(* IEC 61131-3 sources: plcc/tests/fixtures/codegen, 11 files *)

(* ---- function_blocks.st ---- *)
FUNCTION_BLOCK Counter
VAR_INPUT reset : BOOL; END_VAR
VAR_OUTPUT count : INT; END_VAR
VAR cnt : INT := 0; END_VAR
    IF reset THEN cnt := 0; ELSE cnt := cnt + 1; END_IF;
    count := cnt;
END_FUNCTION_BLOCK

FUNCTION_BLOCK Doubler
VAR_INPUT val : INT; END_VAR
VAR_OUTPUT result : INT; END_VAR
    result := val + val;
END_FUNCTION_BLOCK

PROGRAM FBTest
VAR
    c1 : Counter;
    c2 : Counter;
    d : Doubler;
    sum : INT;
    doubled : INT;
END_VAR
    c1(reset := FALSE);
    c2(reset := FALSE);
    d(val := c1.count);
    sum := c1.count + c2.count;
    doubled := d.result;
END_PROGRAM

(* ---- oop.st ---- *)
FUNCTION_BLOCK Accumulator
VAR
    total : INT := 0;
END_VAR
    METHOD Add
    VAR_INPUT val : INT; END_VAR
        total := total + val;
    END_METHOD
    METHOD GetTotal : INT
        GetTotal := total;
    END_METHOD
    METHOD Reset
        total := 0;
    END_METHOD
END_FUNCTION_BLOCK

PROGRAM OOPTest
VAR
    acc : Accumulator;
    result : INT;
END_VAR
    acc.Add(val := 10);
    acc.Add(val := 20);
    acc.Add(val := 30);
    result := acc.GetTotal();
END_PROGRAM

(* ---- arithmetic.st ---- *)
PROGRAM ArithTest
VAR
    a : INT := 0;
    b : INT := 0;
    c : INT := 0;
    d : INT := 0;
    e : INT := 0;
END_VAR
    a := 10 + 5;
    b := 10 - 3;
    c := 4 * 7;
    d := 20 / 4;
    e := 17 MOD 5;
END_PROGRAM

(* ---- arrays_structs.st ---- *)
PROGRAM ArrayTest
VAR
    arr : ARRAY[0..9] OF INT;
    i : INT;
    sum : INT := 0;
    max_val : INT := 0;
END_VAR
    (* Fill array *)
    FOR i := 0 TO 9 DO
        arr[i] := (i + 1) * 10;
    END_FOR;

    (* Sum and find max *)
    sum := 0;
    max_val := arr[0];
    FOR i := 0 TO 9 DO
        sum := sum + arr[i];
        IF arr[i] > max_val THEN max_val := arr[i]; END_IF;
    END_FOR;
END_PROGRAM

(* ---- control_flow.st ---- *)
PROGRAM ControlFlow
VAR
    state : INT := 0;
    output : INT := 0;
    i : INT;
    sum : INT := 0;
END_VAR
    IF state = 0 THEN
        output := 1;
    ELSIF state = 1 THEN
        output := 2;
    ELSE
        output := 3;
    END_IF;

    sum := 0;
    FOR i := 1 TO 10 DO
        sum := sum + i;
    END_FOR;

    WHILE sum > 50 DO
        sum := sum - 10;
    END_WHILE;

    CASE state OF
        0: output := 100;
        1: output := 200;
    ELSE
        output := 0;
    END_CASE;
END_PROGRAM

(* ---- function_calls.st ---- *)
FUNCTION AddTwo : INT
VAR_INPUT
    a : INT;
    b : INT;
END_VAR
    AddTwo := a + b;
END_FUNCTION

FUNCTION Square : INT
VAR_INPUT
    x : INT;
END_VAR
    Square := x * x;
END_FUNCTION

PROGRAM CallTest
VAR
    result1 : INT;
    result2 : INT;
END_VAR
    result1 := AddTwo(3, 4);
    result2 := Square(5);
END_PROGRAM

(* ---- globals.st ---- *)
VAR_GLOBAL
    g_counter : INT;
    g_flag : BOOL;
END_VAR

PROGRAM GlobalTest
VAR
    local_copy : INT;
END_VAR
    g_counter := g_counter + 1;
    local_copy := g_counter;
END_PROGRAM

(* ---- real_fpu.st ---- *)
(* REAL arithmetic for the FPU check (crates/plcc-cli/tests/fpu.rs) and the
   Opta hardware check: results land in %M, so `img` shows them.
   %MW10 = REAL_TO_INT(((1.5 + 2.25) * (1.5 * 2.25) + 0.5) * 100) = 1316,
   %MW11 = REAL_TO_INT(SQRT(2.0) * 1000) = 1414. *)
FUNCTION Scale : REAL
VAR_INPUT
    raw : REAL;
    gain : REAL;
    offset : REAL;
END_VAR
    Scale := raw * gain + offset;
END_FUNCTION

PROGRAM Main
VAR
    a AT %MD0 : REAL := 1.5;
    b AT %MD1 : REAL := 2.25;
    sum AT %MD2 : REAL;
    prod AT %MD3 : REAL;
    q AT %MD4 : REAL;
    r AT %MW10 : INT;
    s AT %MW11 : INT;
END_VAR
    sum := a + b;
    prod := a * b;
    q := Scale(raw := sum, gain := prod, offset := 0.5);
    r := REAL_TO_INT(q * 100.0);
    s := REAL_TO_INT(SQRT(2.0) * 1000.0);
END_PROGRAM

(* ---- stdlib_conversions.st ---- *)
PROGRAM ConversionTest
VAR
    i : INT := 42;
    r : REAL;
    d : DINT;
    b : INT;
END_VAR
    r := INT_TO_REAL(i);
    d := INT_TO_DINT(i);
    b := BOOL_TO_INT(TRUE);
END_PROGRAM

(* ---- stdlib_math.st ---- *)
PROGRAM StdlibMathTest
VAR
    sq : REAL;
    ab : REAL;
    sn : REAL;
    cs : REAL;
    ex : REAL;
    lg : REAL;
    fl : REAL;
    cl : REAL;
    mn : REAL;
    mx : REAL;
    lm : REAL;
END_VAR
    sq := SQRT(25.0);
    ab := ABS(-42.0);
    sn := SIN(0.0);
    cs := COS(0.0);
    ex := EXP(0.0);
    lg := LN(1.0);
    fl := FLOOR(3.7);
    cl := CEIL(3.2);
    mn := MIN(5.0, 3.0);
    mx := MAX(5.0, 3.0);
    lm := LIMIT(0.0, -5.0, 100.0);
END_PROGRAM

(* ---- stdlib_time.st ---- *)
PROGRAM TimeTest
VAR
    t1 : TIME := T#100ms;
    t2 : TIME := T#50ms;
    sum_t : TIME;
    diff_t : TIME;
    scaled_t : TIME;
END_VAR
    sum_t := ADD_TIME(t1, t2);
    diff_t := SUB_TIME(t1, t2);
    scaled_t := MUL_TIME(t1, 3);
END_PROGRAM
